(* Logix 5000 project; controller STAT 1756-L72 rev 20.12; software revision 20.04; part 3 of 34 *)

        [136]   // DELTA LVL NAOH TANK
        [137]   // PARAM CHUTE MAXI LVL NAOH
        [138]   // DELTA LVL H2SO4 TANK
        [139]   // PARAM CHUTE MAXI LVL H2SO4
        [140]   // MEMO LVL H2SO4
   N18 : DINT[120] := ([0] := 2829, [1] := 2829, [2] := 2845, [3] := 2845, [4] := 2829, [5] := 2845, [6] := 2845, [7] := 2845, [8] := 2829, [9] := 2829, [10] := 2845, [11] := 2845, [12] := 2845, [13] := 2845, [14] := 2845, [15] := 2845, [16] := 2845, [17] := 2845, [18] := 2829, [19] := 2820, [20] := 2845, [21] := 2845, [22] := 2845, [23] := 2845, [24] := 781, [25] := 2845, [26] := 781, [27] := 2845, [28] := 2829, [29] := 2820, [30] := 2845, [31] := 2829, [32] := 2829, [33] := 781, [34] := 2829, [35] := 781, [36] := 2829, [37] := 781, [38] := 2829, [39] := 2820, [40] := 2845, [41] := 781, [42] := 2829, [43] := 781, [44] := 2829, [45] := 2829, [46] := 2829, [47] := 2829, [48] := 2829, [49] := 2829, [50] := 2845, [51] := 2844, [52] := 2845, [53] := 2845, [54] := 2845, [55] := 2845, [56] := 2845, [57] := 2845, [58] := 2845, [59] := 2820,
        [60] := 2820, [61] := 2820, [62] := 2820, [63] := 2820, [64] := 2820, [65] := 2820, [66] := 2820, [67] := 2820, [68] := 2820, [69] := 2820, [70] := 2820, [71] := 2820, [72] := 2820, [73] := 2820, [74] := 2820, [75] := 2820, [76] := 2820, [77] := 2820, [78] := 2820, [79] := 2820, [80] := 2820, [105] := -1, [106] := -16369);
   N19 : DINT[80] := ([0] := 1779, [1] := 2603, [2] := 4997, [3] := 7884, [12] := 21845, [14] := 24576, [16] := 2048, [17] := 2048, [18] := 2048, [19] := 2048, [21] := -9, [50] := 128, [51] := 6, [52] := 300, [53] := -32768, [54] := 6, [55] := 300, [60] := 25600, [61] := 6, [62] := 300, [65] := 6, [66] := 300);
   N20 : DINT[80] := ([0] := 7500, [1] := 8000, [2] := 25600, [3] := 8000, [10] := -32768, [11] := 7500, [12] := 8000, [13] := 25600, [14] := 7500, [15] := 26214, [16] := 24576, [17] := 2048, [18] := 2048, [19] := 2048, [21] := -9, [50] := -32640, [51] := 6, [52] := 20, [54] := 7, [55] := 20, [60] := 17408, [62] := 20, [65] := 7, [66] := 20);
   N21 : DINT[80] := ([0] := 8000, [1] := 7000, [2] := 5000, [3] := 3000, [10] := -32768, [11] := 7500, [12] := 8000, [13] := 8000, [14] := 3000, [15] := 26214, [16] := 24576, [17] := 2048, [18] := 2048, [19] := 2048, [21] := -7, [50] := -32640, [51] := 6, [52] := 30, [54] := 7, [55] := 30, [60] := 1024, [62] := 30, [65] := 7, [66] := 30);
   N22 : DINT[80] := ([0] := 24000, [1] := 2000, [2] := 3000, [3] := 32000, [10] := -32768, [11] := 24000, [12] := 2000, [13] := 3000, [14] := 32000, [15] := 8738, [16] := 24576, [17] := 2048, [18] := 2048, [19] := 2048, [21] := -9, [50] := 128, [51] := 6, [52] := 40, [53] := -32768, [54] := 7, [55] := 40, [61] := 6, [62] := 40, [64] := 17408, [66] := 40);
   N23 : DINT[80] := ([0] := 5995, [1] := -2500, [2] := -2500, [3] := -2500, [10] := -32768, [11] := 32000, [12] := 21845, [14] := 24576, [16] := 2048, [17] := 2048, [18] := 2048, [19] := 2048, [21] := -9, [50] := -32640, [51] := 6, [52] := 150, [54] := 6, [55] := 150, [60] := 17408, [62] := 150, [65] := 6, [66] := 150);
        [0]   // DEBIET_PROMAG_33 debiet promag 33 0 -- 10 V
        [1]   // IST_FREQREG_PD1 istt freqreg pd1 0 -- 10 V
        [2]   // IST_FREQREG_PD2 istt freqreg pd2 0 -- 10 V
        [3]   // RESERVE_ANALO_IN reserve analoog ingang 0 tot 10V
   N24 : DINT[80] := ([2] := 234, [3] := 30000, [10] := -32768, [13] := 234, [14] := 30000, [15] := 8738, [16] := 24576, [17] := 2048, [18] := 2048, [19] := 2048, [21] := -9, [50] := -32640, [51] := 6, [52] := 160, [54] := 7, [55] := 160, [61] := 6, [62] := 160, [64] := 25600, [65] := 7, [66] := 160);
        [10]   // ??
        [11]   // SOLL_FREQREG_PD1 soll waarde pd1 0 - 10v
        [12]   // SOLL_FREQREG_PD2 soll freqreg pd2 0 -- 10v
   N26 : DINT[256] := ([0] := 3, [1] := 3, [2] := 7, [3] := 10, [4] := 300, [5] := 900, [6] := 20, [7] := 850, [8] := 60, [9] := 30, [20] := 2, [21] := 2, [22] := 7, [23] := 10, [24] := 300, [25] := 900, [26] := 20, [27] := 850, [28] := 60, [29] := 30, [36] := 1764, [42] := 15, [43] := 10, [44] := 30, [45] := 1200, [46] := 1800, [47] := 4500, [48] := 33, [49] := 5, [58] := 35, [62] := 15, [63] := 10, [64] := 30, [65] := 900, [66] := 1800, [67] := 4500, [68] := 33, [69] := 5, [82] := 20, [83] := 60, [84] := 60, [85] := 30, [86] := 120, [87] := 700, [88] := 20, [89] := 850, [90] := 60, [91] := 60, [102] := 15, [103] := 35, [104] := 10, [105] := 900, [106] := 1800, [107] := 4500, [108] := 35, [109] := 5, [122] := 15, [123] := 35, [124] := 10, [125] := 900,
        [126] := 1800, [127] := 4500, [128] := 35, [129] := 5, [132] := 10, [133] := 50, [134] := 10, [135] := 60, [136] := 7, [137] := 7, [138] := 960, [142] := 10, [143] := 50, [144] := 10, [145] := 60, [146] := 7, [148] := 900, [152] := 10, [153] := 50, [154] := 10, [155] := 60, [156] := 7, [158] := 960, [172] := 10, [173] := 1, [174] := 1, [175] := 9000, [176] := 600, [177] := 1, [178] := 1, [179] := 1800, [182] := 20, [183] := 1, [184] := 1, [185] := 18000, [186] := 600, [187] := 1, [188] := 1, [189] := 1800, [190] := 1, [191] := 1, [192] := 5, [193] := 1, [194] := 1, [195] := 1800, [196] := 600, [197] := 1, [198] := 1, [199] := 1800, [200] := 1, [201] := 2000, [202] := 600, [203] := 1, [204] := 1, [205] := 1800, [206] := 600);
        [0]   // SOLL_ST_SPOELTFB75_1 Soll stap spoel TFB 75-1 ingave via visualisatie
        [1]   // IST_ST_SPOELTFB75_1 Ist stap spoel TFB 75-1 ingave via visualisatie
        [2]   // SOLL_TIJD_ST_1 Soll tijd stap 1 spoel TFB75 -1 Afsluiten filter
        [3]   // SOLL_TIJD_ST_2 Soll tijd stap 2 spoel TFB75 -1 Aflaten water
        [4]   // SOLL_TIJD_ST_3 Soll tijd stap 3 spoel TFB75 -1 luchtspoeling
        [5]   // SOLL_TIJD_ST_4 Soll tijd stap 4 spoel TFB75 -1 rustpauze
        [6]   // SOLL_TIJD_ST_5 Soll tijd stap 5 spoel TFB75 -1 Waterspoeling
        [7]   // SOLL_TIJD_ST_6 Soll tijd stap 6 spoel TFB75 -1 Rustpauze
        [8]   // SOLL_TIJD_ST_7 Soll tijd stap 7 spoel TFB75 -1 Openen filter
        [10]   // SOLL_TIJD_ST_8
        [11]   // SOLL_TIJD_ST_9
        [12]   // SOLL_TIJD_ST_10
        [13]   // SOLL_TIJD_ST_11
        [14]   // SOLL_TIJD_ST_12
        [15]   // SOLL_TIJD_ST_13
        [16]   // SOLL_TIJD_ST_14
        [17]   // SOLL_TIJD_ST_15
        [18]   // SOLL_TIJD_ST_16
        [20]   // SOLL_ST_SPOETFB75_2
        [21]   // IST_ST_SPOETFB75_2
        [22]   // SOLL_TIJD_STA_1_1
        [23]   // SOLL_TIJD_STA_2_2
        [24]   // SOLL_TIJD_STA_3_2
        [25]   // SOLL_TIJD_STA_4_2
        [26]   // SOLL_TIJD_STA_5_2
        [27]   // SOLL_TIJD_STA_6_2
        [28]   // SOLL_TIJD_STA_7_2
   N28 : DINT[80] := ([0] := 10249, [1] := 10249, [2] := 10249, [3] := 10249, [10] := -32768, [11] := 32000, [12] := 26214, [14] := 24576, [16] := 2048, [17] := 2048, [18] := 2048, [19] := 2048, [21] := -11, [22] := -11, [50] := 128, [51] := 6, [52] := 150, [53] := -32768, [54] := 6, [55] := 150, [60] := 4096, [62] := 150, [63] := -11, [66] := 150, [67] := -11);
   N7 : DINT[255] := ([0] := 7825, [1] := 3859, [2] := 8045, [3] := -2501, [12] := 21845, [14] := 24576, [16] := 2048, [17] := 2048, [18] := 2048, [19] := 2048, [21] := -9, [33] := 16383, [40] := 45, [41] := 40, [42] := 35, [43] := 50, [44] := 45, [45] := 35, [50] := -32640, [51] := 6, [52] := 260, [54] := 6, [55] := 260, [60] := 17408, [62] := 260, [65] := 6, [66] := 260, [70] := 80, [71] := 38, [72] := 78, [92] := 6, [100] := 15900, [101] := 15900, [110] := -32768, [111] := 4, [186] := 16, [190] := 7, [191] := 1, [197] := 2, [198] := 8, [199] := 96, [200] := 22, [201] := 1564, [211] := 1028, [225] := 1048576, [234] := 31233);
        [70]   // aux LEVEL TANK RECUP L3
        [71]   // n7:71
        [90]   // ?
        [97]   // ?
        [98]   // ?
        [111]   // HULPWOORD_N1
        [112]   // HULPWOORD_N2
        [113]   // HULPWOORD_N3
        [114]   // HULPWOORD_N4
        [115]   // HULPWOORD_N5
        [190]   // PRIORITE DEFAUT
        [191]   // defaut niv 2
        [197]   // NOMBRE DEFAUT EXISTANT ACQUITE
        [198]   // NOMBRE NOUVEAU DEFAUT
        [199].0   // arret entretien
        [199].1   // acquit defaut
        [199].5   // new defaut
        [199].6   // ancien defaut present
        [200].0   // PMP ETANG EN DEF
        [200].1   // no flow pumping from etang
        [200].2   // FLOW TOO LOW Q1
        [200].3   // LEVEL PRETREATED TOO HIGH
        [200].4   // LEVEL LOW PRETREATED WATER WARNING
        [200].5   // LEVEL LOW PRETREATED WATER
        [200].6   // ANORMAL EMPTYING PRETREATED WATER TANK
        [200].7   // 2 pump pretreated tank out of order P3&P4
        [200].8   // no flow pumping from PRETREATED WATER TANK
        [200].9   // FLOW TOO LOW Q2
        [200].11   // recup water tank L1 too high
        [200].12   // PMP RECUP L1 OUT OF ORDER
        [200].13   // recup water tank L2 too high
        [200].14   // PMP RECUP L2 OUT OF ORDER
        [200].15   // recup water tank L3 too high
        [201].0   // PMP RECUP L3 OUT OF ORDER
        [201].1   // recup water tank L4 too high
        [201].2   // PMP RECUP L4 OUT OF ORDER
        [201].3   // LEVEL NAOH TOO HIGH
        [201].4   // ANORMAL LEVEL DECREASE naoh TANK
        [201].5   // LACK DETECTIE NAOH
        [201].6   // LEVEL H2SO4 TOO HIGH
        [201].7   // ANORMAL LEVEL DECREASE H2SO4 TANK
        [201].8   // LACK DETECTIE H2SO4
        [201].9   // defaut niveau vijver trop bas
        [201].10   // defaut niveau puisard ligne 4
        [201].11   // defaut vanne position eau ville
        [210].0   // PMP ETANG EN DEF
        [210].1   // no flow pumping from etang
        [210].2   // FLOW TOO LOW Q1
        [210].3   // LEVEL PRETREATED TOO HIGH
        [210].4   // LEVEL LOW PRETREATED WATER WARNING
        [210].5   // LEVEL LOW PRETREATED WATER
        [210].6   // ANORMAL EMPTYING PRETREATED WATER TANK
        [210].7   // 2 pump pretreated tank out of order P3&P4
        [210].8   // no flow pumping from PRETREATED WATER TANK
        [210].9   // FLOW TOO LOW Q2
        [210].11   // recup water tank L1 too high
        [210].12   // PMP RECUP L1 OUT OF ORDER
        [210].13   // recup water tank L2 too high
        [210].14   // PMP RECUP L2 OUT OF ORDER
        [210].15   // recup water tank L3 too high
        [211].0   // PMP RECUP L3 OUT OF ORDER
        [211].1   // recup water tank L4 too high
        [211].2   // PMP RECUP L4 OUT OF ORDER
        [211].3   // LEVEL NAOH TOO HIGH
        [211].4   // ANORMAL LEVEL DECREASE naoh TANK
        [211].5   // LACK DETECTIE NAOH
        [211].6   // LEVEL H2SO4 TOO HIGH
        [211].7   // ANORMAL LEVEL DECREASE H2SO4 TANK
        [211].8   // LACK DETECTIE H2SO4
        [211].9   // defaut niveau vijver trop bas
        [211].11   // memo defaut vanne position eau ville
   N7_70 : REAL := 80.299995;
   N7_71 : REAL := 99.04;
   N7_72 : REAL := 1561.2001;
   naohL1VA4 : BOOL;
   naohL2VA4 : BOOL;
   O1 : INT[32] := ([6] := 2#1000_0000_0000_0000, [11] := 2#0000_0000_0000_0011, [12] := 2#0000_0000_0000_0010, [20] := 2#0000_0110_0000_0110);
   O11 : INT[2] := ([0] := 2#0101_1000_0001_1010, [1] := 2#1011_0000_0000_0110);
   O11_000_Bit00 : ALIAS FOR O11[0].0;   // Motor P11 lijn 1 P11_LIJN_1
   O11_000_Bit01 : ALIAS FOR O11[0].1;   // Motor P12 lijn 1 P12_LIJN_1
   O11_000_Bit02 : ALIAS FOR O11[0].2;   // Motor P13 lijn 2 P13_LIJN_2
   O11_000_Bit03 : ALIAS FOR O11[0].3;   // Motor P14 lijn 2 P14_LIJN_2
   O11_000_Bit04 : ALIAS FOR O11[0].4;   // Motor P15 lijn 3 P15_LIJN_3
   O11_000_Bit05 : ALIAS FOR O11[0].5;   // Motor P16 lijn 3 P16_LIJN_3
   O11_000_Bit06 : ALIAS FOR O11[0].6;   // Motor P17 lijn 4 P17_LIJN_4
   O11_000_Bit07 : ALIAS FOR O11[0].7;   // Motor P18 lijn 4 P18_LIJN_4
   O11_000_Bit08 : ALIAS FOR O11[0].8;   // Pomp voeding osmose 1 lijn PRO1_OSMO1_LIJN
   O11_000_Bit09 : ALIAS FOR O11[0].9;   // Pomp voeding osmose 1 driehoek PRO1_OSMO1_DRIE
   O11_000_Bit10 : ALIAS FOR O11[0].10;   // Pomp voeding osmose 1 ster PRO1_OSMO1_STER
   O11_000_Bit11 : ALIAS FOR O11[0].11;   // Pomp voeding osmose 2 lijn PRO1_OSMO2_LIJN
   O11_000_Bit12 : ALIAS FOR O11[0].12;   // Pomp voeding osmose 2 driehoek PRO1_OSMO2_DRIE
   O11_000_Bit13 : ALIAS FOR O11[0].13;   // Pomp voeding osmose 2 ster PRO1_OSMO2_STER
   O11_000_Bit14 : ALIAS FOR O11[0].14;   // pomp 21 kuip az P21_KUIP_AZ_LIJN
   O11_000_Bit15 : ALIAS FOR O11[0].15;   // pomp p21 kuip az driehoek P21_KUIP_AZ_DRIE
   O11_001_Bit00 : ALIAS FOR O11[1].0;   // pomp p21 kuip az ster P21_KUIP_AZ_STER
   O11_001_Bit01 : ALIAS FOR O11[1].1;   // pomp p22 kuip az lijn P22_KUIP_AZ_LIJN
   O11_001_Bit02 : ALIAS FOR O11[1].2;   // pomp p22 kuip az drie P22_KUIP_AZ_DRIE
   O11_001_Bit03 : ALIAS FOR O11[1].3;   // pomp p22 kuip az ster P22_KUIP_AZ_STER
   O11_001_Bit04 : ALIAS FOR O11[1].4;   // Voedingspomp osmose 3 in lijn PRO3_OSMOSE3_LIJN
   O11_001_Bit05 : ALIAS FOR O11[1].5;   // Voedingspomp osmose 3 in drie PRO3_OSMOSE3_DRIE
   O11_001_Bit06 : ALIAS FOR O11[1].6;   // Voedingspomp osmose 3 in ster PRO3_OSMOSE3_STER
   O11_001_Bit07 : ALIAS FOR O11[1].7;   // reinigingspomp membraam P21_REINIG
   O11_001_Bit08 : ALIAS FOR O11[1].8;   // ventilator s1 S1_VENT
   O11_001_Bit09 : ALIAS FOR O11[1].9;   // pomp voeding drive 1 in lijn P3_FAB_LIJN
   O11_001_Bit10 : ALIAS FOR O11[1].10;   // pomp debloquage 1 P3 P3_FAB_DRIE
   O11_001_Bit11 : ALIAS FOR O11[1].11;   // pomp voeding fab1 in ster P3_FAB_STER
   O11_001_Bit12 : ALIAS FOR O11[1].12;   // pomp voeding fabriek 2 in lijn P4_FAB_LIJN
   O11_001_Bit13 : ALIAS FOR O11[1].13;   // deverouillage drive P4 P4_FAB_DRIE
   O11_001_Bit14 : ALIAS FOR O11[1].14;   // reserve P4_FAB_STER
   O11_001_Bit15 : ALIAS FOR O11[1].15;   // spoelpomp filters dubbele media P5_SPOEL
   O12 : INT[2] := ([0] := 2#1100_1000_1001_1000, [1] := 2#0111_0100_1101_0000);
   O12_000_Bit00 : ALIAS FOR O12[0].0;   // spoelpomp filters dubbele media P6_SPOEL
   O12_000_Bit01 : ALIAS FOR O12[0].1;   // pomp pompen uit kelder P23_KELDER
   O12_000_Bit02 : ALIAS FOR O12[0].2;   // pomp pompen uit kelder P24_KELDER
   O12_000_Bit03 : ALIAS FOR O12[0].3;   // motor ag1 mixer krimp neutralisatie AG1_MIXER_KRIMP
   O12_000_Bit04 : ALIAS FOR O12[0].4;   // Motor doseerpomp acide pd3 PD3_DOS_ACIDE
   O12_000_Bit05 : ALIAS FOR O12[0].5;   // Motor doseerpomp acide pd4 PD4_DOS_ACIDE
   O12_000_Bit06 : ALIAS FOR O12[0].6;   // Motor doseerpomp acide pd5 soude PD5_DOS_SOUDE
   O12_000_Bit07 : ALIAS FOR O12[0].7;   // Motor doseerpomp acide pd6 soude PD6_DOS_SOUDE
   O12_000_Bit08 : ALIAS FOR O12[0].8;   // pomp ag2 mixer vat 1 AG2_MIXER_VAT1
   O12_000_Bit09 : ALIAS FOR O12[0].9;   // pomp ag3 mixer vat 2 AG3_MIXER_VAT2
   O12_000_Bit10 : ALIAS FOR O12[0].10;   // pomp pd7 doseerpomp floculaat PD7_DOSEER_FLOCU
   O12_000_Bit11 : ALIAS FOR O12[0].11;   // pomp pd8 doseerpomp floculaat PD8_DOSEER_FLOCU
   O12_000_Bit12 : ALIAS FOR O12[0].12;   // Motor P19a zuiveringspomp controleweger P19_ZUIVERP
   O12_000_Bit13 : ALIAS FOR O12[0].13;   // Motor P20 zuiveringspomp controleweger P20_ZUIVERP
   O12_000_Bit14 : ALIAS FOR O12[0].14;   // Motor Pm1 recerculatiepomp ingang 1 decanter PM1_RECER_DEC1
   O12_000_Bit15 : ALIAS FOR O12[0].15;   // Motor Pm2 recerculatiepomp ingang 2 decanter PM2_RECER_DEC2
   O12_001_Bit00 : ALIAS FOR O12[1].0;   // Motor Pm3 evacuatiepomp ingang 1 decanter PM3_EVACU_IN_1
   O12_001_Bit01 : ALIAS FOR O12[1].1;   // Motor Pm4 evacuatiepomp ingang 2 decanter PM4_EVACU_IN_2
   O12_001_Bit02 : ALIAS FOR O12[1].2;   // Motor P25 pekel P25_POMP_PEKEL
   O12_001_Bit03 : ALIAS FOR O12[1].3;   // Motor P7 voedingspomp omgekeerde osmose 1 P7_OSMOSE_1
   O12_001_Bit04 : ALIAS FOR O12[1].4;   // Motor P8 voedingspomp omgekeerde osmose 2 P8_OSMOSE_2
   O12_001_Bit05 : ALIAS FOR O12[1].5;   // Motor P9 voedingspomp omgekeerde osmose 3 P9_OSMOSE_3
   O12_001_Bit06 : ALIAS FOR O12[1].6;   // TFB1_1_EV1 TFB1_1_EV1
   O12_001_Bit07 : ALIAS FOR O12[1].7;   // TFB1_1_EV2 TFB1_1_EV2
   O12_001_Bit08 : ALIAS FOR O12[1].8;   // TFB1_2_EV3 TFB1_2_EV3
   O12_001_Bit09 : ALIAS FOR O12[1].9;   // TFB1_2_EV4 TFB1_2_EV4
   O12_001_Bit10 : ALIAS FOR O12[1].10;   // TFB1_2_EV10 TFB1_2_EV10
   O12_001_Bit11 : ALIAS FOR O12[1].11;   // TFB1_EV9 TFB1_EV9
   O12_001_Bit12 : ALIAS FOR O12[1].12;   // TFB1_2_EV5 TFB1_2_EV5
   O12_001_Bit13 : ALIAS FOR O12[1].13;   // TFB1_2_EV6 TFB1_2_EV6
   O12_001_Bit14 : ALIAS FOR O12[1].14;   // STFA1_EV1 STFA1_EV1
   O12_001_Bit15 : ALIAS FOR O12[1].15;   // STFA1_EV2 STFA1_EV2
   O13 : INT[2] := ([0] := 2#0000_0000_0000_1000, [1] := 2#0001_0000_0000_0000);
   O13_000_Bit00 : ALIAS FOR O13[0].0;   // STFA1_EV3 STFA1_EV3
   O13_000_Bit01 : ALIAS FOR O13[0].1;   // STFA1_EV4 STFA1_EV4
   O13_000_Bit02 : ALIAS FOR O13[0].2;   // STFA1_EV5 STFA1_EV5
   O13_000_Bit03 : ALIAS FOR O13[0].3;   // STFA1_EV6 STFA1_EV6
   O13_000_Bit06 : ALIAS FOR O13[0].6;   // PULS_DOSEER_PD3
   O13_000_Bit07 : ALIAS FOR O13[0].7;   // PULS_DOSEER_PD4
   O13_000_Bit08 : ALIAS FOR O13[0].8;   // PULS_DOSEER_PD5
   O13_000_Bit09 : ALIAS FOR O13[0].9;   // PULS_DOSEER_PD6
   O13_000_Bit12 : ALIAS FOR O13[0].12;   // STFA2_EV1 STFA2_EV1
   O13_000_Bit13 : ALIAS FOR O13[0].13;   // STFA2_EV2 STFA2_EV2
   O13_000_Bit14 : ALIAS FOR O13[0].14;   // STFA2_EV3 STFA2_EV3
   O13_000_Bit15 : ALIAS FOR O13[0].15;   // STFA2_EV4 STFA2_EV4
   O13_001_Bit0 : ALIAS FOR O13[1].0;   // STFA2_EV5 STFA2_EV5
   O13_001_Bit1 : ALIAS FOR O13[1].1;   // STFA2_EV6 STFA2_EV6
   O13_001_Bit10 : ALIAS FOR O13[1].10;   // TFB1_2_EV7 TFB1_2_EV7
   O13_001_Bit11 : ALIAS FOR O13[1].11;   // TFB1_2_EV8 TFB1_2_EV8
   O13_001_Bit12 : ALIAS FOR O13[1].12;   // TFB1_2_EV11 TFB1_2_EV11
   O13_001_Bit13 : ALIAS FOR O13[1].13;   // vanne eau de ville
   O14 : INT[2] := ([0] := 2#1000_0000_0000_0000, [1] := 2#0011_0000_0010_0010);
   O14_000_Bit14 : ALIAS FOR O14[0].14;   // STFA3_EV1 STFA3_EV1
   O14_000_Bit15 : ALIAS FOR O14[0].15;   // STFA3_EV2 STFA3_EV2
   O14_001_Bit00 : ALIAS FOR O14[1].0;   // STFA3_EV3 STFA3_EV3
   O14_001_Bit01 : ALIAS FOR O14[1].1;   // STFA3_EV4 STFA3_EV4
   O14_001_Bit02 : ALIAS FOR O14[1].2;   // STFA3_EV5 STFA3_EV5
   O14_001_Bit03 : ALIAS FOR O14[1].3;   // STFA3_EV6 STFA3_EV6
   O14_001_Bit04 : ALIAS FOR O14[1].4;   // kalxon out NAOH
   O14_001_Bit05 : ALIAS FOR O14[1].5;   // lampe out NAOH
   O14_001_Bit06 : ALIAS FOR O14[1].6;   // klaxon out H2SO4
   O14_001_Bit07 : ALIAS FOR O14[1].7;   // lampe H2SO4
   O14_001_Bit08 : ALIAS FOR O14[1].8;   // klaxon out ZOUT
   O14_001_Bit09 : ALIAS FOR O14[1].9;   // lampe ZOUT
   O14_001_Bit12 : ALIAS FOR O14[1].12;   // RO1_EV1 RO1_EV1
   O14_001_Bit13 : ALIAS FOR O14[1].13;   // RO1_EV2 RO1_EV2
   O15 : INT[2] := ([1] := 2#0000_0000_1000_0000);
   O15_000_Bit00 : ALIAS FOR O15[0].0;   // RO2_EV1 RO2_EV1
   O15_000_Bit01 : ALIAS FOR O15[0].1;   // RO2_EV2 RO2_EV2
   O15_000_Bit04 : ALIAS FOR O15[0].4;   // RO3_EV1 RO3_EV1
   O15_000_Bit05 : ALIAS FOR O15[0].5;   // RO3_EV2 RO3_EV2
   O15_000_Bit09 : ALIAS FOR O15[0].9;   // CLEAN_V11 CLEAN_V11
   O15_000_Bit10 : ALIAS FOR O15[0].10;   // CLEAN_V12 CLEAN_V12
   O15_000_Bit11 : ALIAS FOR O15[0].11;   // CLEAN_V13 CLEAN_V13
   O15_000_Bit12 : ALIAS FOR O15[0].12;   // CLEAN_V14 CLEAN_V14
   O15_000_Bit13 : ALIAS FOR O15[0].13;   // CLEAN_V21 CLEAN_V21
   O15_000_Bit14 : ALIAS FOR O15[0].14;   // CLEAN_V22 CLEAN_V22
   O15_000_Bit15 : ALIAS FOR O15[0].15;   // CLEAN_V23 CLEAN_V23
   O15_001_Bit00 : ALIAS FOR O15[1].0;   // CLEAN_V24 CLEAN_V24
   O15_001_Bit01 : ALIAS FOR O15[1].1;   // CLEAN_V3 CLEAN_V3
   O15_001_Bit06 : ALIAS FOR O15[1].6;   // EV2 EV2
   O15_001_Bit07 : ALIAS FOR O15[1].7;   // EV3 EV3
   O15_001_Bit08 : ALIAS FOR O15[1].8;   // EV4 EV4
   O15_001_Bit09 : ALIAS FOR O15[1].9;   // EV5 EV5
   O15_001_Bit10 : ALIAS FOR O15[1].10;   // EV6 EV6
   O15_001_Bit11 : ALIAS FOR O15[1].11;   // EV7 EV7
   O15_001_Bit13 : ALIAS FOR O15[1].13;   // TFB2_1_EV1 TFB2_1_EV1
   O15_001_Bit14 : ALIAS FOR O15[1].14;   // TFB2_1_EV2 TFB2_1_EV2
   O15_001_Bit15 : ALIAS FOR O15[1].15;   // TFB2_1_EV3 TFB2_1_EV3
   O16 : INT[2] := ([0] := 2#1001_0100_0000_1001, [1] := 2#1100_0000_0000_0000);
        [0].4   // vanne soude de stock
        [0].3   // vanne ibt acide de stock
   O16_000_Bit00 : ALIAS FOR O16[0].0;   // COMMANDE VANNE ALIBERT
   O16_000_Bit01 : ALIAS FOR O16[0].1;   // vanne pmp puit 3
   O16_000_Bit02 : ALIAS FOR O16[0].2;   // vanne pmp puit 2
   O16_000_Bit03 : ALIAS FOR O16[0].3;
   O16_000_Bit09 : ALIAS FOR O16[0].9;   // LAMP_P17_AAN
   O16_000_Bit10 : ALIAS FOR O16[0].10;   // LAMP_P17_UIT
   O16_000_Bit11 : ALIAS FOR O16[0].11;   // LAMP_P18_AAN
   O16_000_Bit12 : ALIAS FOR O16[0].12;   // LAMP_P18_UIT
   O16_000_Bit15 : ALIAS FOR O16[0].15;   // LAMP_PRO1_AAN
   O16_001_Bit00 : ALIAS FOR O16[1].0;   // LAMP_PRO1_UIT
   O16_001_Bit01 : ALIAS FOR O16[1].1;   // LAMP_PRO2_AAN
   O16_001_Bit02 : ALIAS FOR O16[1].2;   // LAMP_PRO2_UIT
   O16_001_Bit03 : ALIAS FOR O16[1].3;   // LAMP_P21_AAN
   O16_001_Bit04 : ALIAS FOR O16[1].4;   // LAMP_P21_UIT
   O16_001_Bit05 : ALIAS FOR O16[1].5;   // LAMP_P22_AAN
   O16_001_Bit06 : ALIAS FOR O16[1].6;   // LAMP_P22_UIT
   O16_001_Bit07 : ALIAS FOR O16[1].7;   // LAMP_PRO3_AAN
   O16_001_Bit08 : ALIAS FOR O16[1].8;   // LAMP_PRO3_UIT
   O16_001_Bit09 : ALIAS FOR O16[1].9;   // LAMP_P21_REINIG_AAN
   O16_001_Bit10 : ALIAS FOR O16[1].10;   // LAMP_P21_REINIG_UIT
   O16_001_Bit11 : ALIAS FOR O16[1].11;   // LAMP_VENT_S1_AAN
   O16_001_Bit12 : ALIAS FOR O16[1].12;   // LAMP_VENT_S1_UIT
   O16_001_Bit13 : ALIAS FOR O16[1].13;   // LAMP_P3_AAN
   O16_001_Bit14 : ALIAS FOR O16[1].14;   // LAMP_P3_UIT
   O16_001_Bit15 : ALIAS FOR O16[1].15;   // LAMP_P4_AAN
   O17 : INT[2] := ([0] := 2#0000_0010_0000_0000, [1] := 2#0010_1010_0001_0010);
   O17_000_Bit00 : ALIAS FOR O17[0].0;   // LAMP_P4_UIT
   O17_000_Bit01 : ALIAS FOR O17[0].1;   // LAMP_P5_AAN
   O17_000_Bit02 : ALIAS FOR O17[0].2;   // LAMP_P5_UIT
   O17_000_Bit03 : ALIAS FOR O17[0].3;   // LAMP_P6_AAN
   O17_000_Bit04 : ALIAS FOR O17[0].4;   // LAMP_P6_UIT
   O17_000_Bit05 : ALIAS FOR O17[0].5;   // LAMP_P23_AAN
   O17_000_Bit06 : ALIAS FOR O17[0].6;   // LAMP_P23_UIT
   O17_000_Bit07 : ALIAS FOR O17[0].7;   // LAMP_P24_AAN
   O17_000_Bit08 : ALIAS FOR O17[0].8;   // LAMP_P24_UIT
   O17_000_Bit09 : ALIAS FOR O17[0].9;   // LAMP_AG1_AAN
   O17_000_Bit10 : ALIAS FOR O17[0].10;   // LAMP_AG1_UIT
   O17_000_Bit11 : ALIAS FOR O17[0].11;   // LAMP_AG2_AAN
   O17_000_Bit12 : ALIAS FOR O17[0].12;   // LAMP_AG2_UIT
   O17_000_Bit13 : ALIAS FOR O17[0].13;   // LAMP_AG3_AAN
   O17_000_Bit14 : ALIAS FOR O17[0].14;   // LAMP_AG3_UIT
   O17_000_Bit15 : ALIAS FOR O17[0].15;   // LAMP_PD7_AAN
   O17_001_Bit00 : ALIAS FOR O17[1].0;   // LAMP_PD7_UIT
   O17_001_Bit01 : ALIAS FOR O17[1].1;   // LAMP_PD8_AAN
   O17_001_Bit02 : ALIAS FOR O17[1].2;   // LAMP_PD8_UIT
   O17_001_Bit03 : ALIAS FOR O17[1].3;   // LAMP_P19A_AAN
   O17_001_Bit04 : ALIAS FOR O17[1].4;   // LAMP_P19A_UIT
   O17_001_Bit05 : ALIAS FOR O17[1].5;   // LAMP_P19B_AAN
   O17_001_Bit06 : ALIAS FOR O17[1].6;   // LAMP_P19B_UIT
   O17_001_Bit09 : ALIAS FOR O17[1].9;   // LAMP_P25_AAN
   O17_001_Bit10 : ALIAS FOR O17[1].10;   // LAMP_P25_UIT
   O17_001_Bit11 : ALIAS FOR O17[1].11;   // LAMP_PM1_AAN
   O17_001_Bit12 : ALIAS FOR O17[1].12;   // LAMP_PM1_UIT
   O17_001_Bit13 : ALIAS FOR O17[1].13;   // LAMP_PM2_AAN
   O17_001_Bit14 : ALIAS FOR O17[1].14;   // LAMP_PM2_UIT
   O17_001_Bit15 : ALIAS FOR O17[1].15;   // LAMP_PM3_AAN
   O18 : INT[2] := ([0] := 2#0000_0010_0000_0000, [1] := 2#0000_0000_0001_0100);
   O18_000_Bit00 : ALIAS FOR O18[0].0;   // LAMP_PM3_UIT
   O18_000_Bit01 : ALIAS FOR O18[0].1;   // LAMP_PM4_AAN
   O18_000_Bit02 : ALIAS FOR O18[0].2;   // LAMP_PM4_UIT
   O18_000_Bit07 : ALIAS FOR O18[0].7;   // LAMP_P7_AAN
   O18_000_Bit08 : ALIAS FOR O18[0].8;   // LAMP_P7_UIT
   O18_000_Bit09 : ALIAS FOR O18[0].9;   // LAMP_P8_AAN
   O18_000_Bit10 : ALIAS FOR O18[0].10;   // LAMP_P8_UIT
   O18_000_Bit11 : ALIAS FOR O18[0].11;   // LAMP_P9_AAN
   O18_000_Bit12 : ALIAS FOR O18[0].12;   // LAMP_P9_UIT
   O18_001_Bit00 : ALIAS FOR O18[1].0;   // pompe 1 puisard ligne 4
   O18_001_Bit01 : ALIAS FOR O18[1].1;   // pompe 2 puisard ligne 4
   O18_001_Bit02 : ALIAS FOR O18[1].2;   // pmp put 2
   O18_001_Bit03 : ALIAS FOR O18[1].3;   // PMP PUT over
   O18_001_Bit04 : ALIAS FOR O18[1].4;   // PMP PUT 1
   O18_001_Bit05 : ALIAS FOR O18[1].5;   // pmp vijver IWM
   O18_001_Bit06 : ALIAS FOR O18[1].6;
   O18_001_Bit07 : ALIAS FOR O18[1].7;   // pomp pompen uit kelder p23
   O18_001_Bit08 : ALIAS FOR O18[1].8;   // pomp pompen uit kelder p24
   O1_006_Bit15 : ALIAS FOR O1[6].15;
   O1_011_Bit00 : ALIAS FOR O1[11].0;
   O1_011_Bit01 : ALIAS FOR O1[11].1;
   O1_011_Bit02 : ALIAS FOR O1[11].2;
   O1_011_Bit03 : ALIAS FOR O1[11].3;
   O1_011_Bit04 : ALIAS FOR O1[11].4;
   O1_011_Bit05 : ALIAS FOR O1[11].5;
   O1_011_Bit06 : ALIAS FOR O1[11].6;
   O1_011_Bit07 : ALIAS FOR O1[11].7;
   O1_011_Bit08 : ALIAS FOR O1[11].8;
   O1_011_Bit09 : ALIAS FOR O1[11].9;
   O1_011_Bit10 : ALIAS FOR O1[11].10;
   O1_012_Bit01 : ALIAS FOR O1[12].1;
   O1_012_Bit02 : ALIAS FOR O1[12].2;
   O1_012_Bit03 : ALIAS FOR O1[12].3;
   O1_012_Bit04 : ALIAS FOR O1[12].4;
   O1_012_Bit05 : ALIAS FOR O1[12].5;
   O1_012_Bit06 : ALIAS FOR O1[12].6;
   O1_012_Bit07 : ALIAS FOR O1[12].7;
   O1_012_Bit08 : ALIAS FOR O1[12].8;
   O1_012_Bit09 : ALIAS FOR O1[12].9;
   O1_012_Bit10 : ALIAS FOR O1[12].10;
   O1_020_Bit00 : ALIAS FOR O1[20].0;
   O1_020_Bit01 : ALIAS FOR O1[20].1;
   O1_020_Bit02 : ALIAS FOR O1[20].2;
   O1_020_Bit03 : ALIAS FOR O1[20].3;
   O1_020_Bit08 : ALIAS FOR O1[20].8;
   O1_020_Bit09 : ALIAS FOR O1[20].9;
   O1_020_Bit10 : ALIAS FOR O1[20].10;
   O1_020_Bit11 : ALIAS FOR O1[20].11;
   O1_021_Bit00 : ALIAS FOR O1[21].0;
   O1_021_Bit01 : ALIAS FOR O1[21].1;
   O1_021_Bit02 : ALIAS FOR O1[21].2;
   O1_021_Bit03 : ALIAS FOR O1[21].3;
   O1_021_Bit08 : ALIAS FOR O1[21].8;
   O1_021_Bit09 : ALIAS FOR O1[21].9;
   O20 : INT[8] := ([0] := 2#0000_1011_0000_1101, [1] := 2#0000_1011_0000_1101, [2] := 2#0000_1011_0001_1101, [3] := 2#0000_1011_0001_1101, [4] := 2#0000_1011_0000_1101, [5] := 2#0000_1011_0001_1101, [6] := 2#0000_1011_0001_1101, [7] := 2#0000_1011_0001_1101);
   O20_000 : ALIAS FOR O20[0];
   O20_001 : ALIAS FOR O20[1];
   O20_002 : ALIAS FOR O20[2];
   O20_003 : ALIAS FOR O20[3];
   O20_004 : ALIAS FOR O20[4];
   O20_005 : ALIAS FOR O20[5];
   O20_006 : ALIAS FOR O20[6];
   O20_007 : ALIAS FOR O20[7];
   O21 : INT[8] := ([0] := 2#0000_1011_0001_1101, [1] := 2#0000_1011_0001_1101, [2] := 2#0000_1011_0001_1101, [3] := 2#0000_1011_0001_1101, [4] := 2#0000_1011_0001_1101, [5] := 2#0000_1011_0001_1101, [6] := 2#0000_1011_0001_1101, [7] := 2#0000_1011_0001_1101);
   O21_000 : ALIAS FOR O21[0];
   O21_001 : ALIAS FOR O21[1];
   O21_002 : ALIAS FOR O21[2];
   O21_003 : ALIAS FOR O21[3];
   O21_004 : ALIAS FOR O21[4];
   O21_005 : ALIAS FOR O21[5];
   O21_006 : ALIAS FOR O21[6];
   O21_007 : ALIAS FOR O21[7];
   O22 : INT[8] := ([0] := 2#0000_1011_0001_1101, [1] := 2#0000_1011_0001_1101, [2] := 2#0000_1011_0001_1101, [3] := 2#0000_1011_0001_1101, [4] := 2#0000_0011_0000_1101, [5] := 2#0000_1011_0001_1101, [6] := 2#0000_0011_0000_1101, [7] := 2#0000_1011_0001_1101);
   O22_000 : ALIAS FOR O22[0];
   O22_000_Bit04 : ALIAS FOR O22[0].4;
   O22_001 : ALIAS FOR O22[1];
   O22_002 : ALIAS FOR O22[2];
   O22_003 : ALIAS FOR O22[3];
   O22_004 : ALIAS FOR O22[4];
   O22_005 : ALIAS FOR O22[5];
   O22_006 : ALIAS FOR O22[6];
   O22_007 : ALIAS FOR O22[7];
   O23 : INT[8] := ([0] := 2#0000_1011_0001_1101, [1] := 2#0000_1011_0000_1101, [2] := 2#0000_1011_0000_1101, [3] := 2#0000_0011_0000_1101, [4] := 2#0000_1011_0000_1101, [5] := 2#0000_1011_0000_1101, [6] := 2#0000_1011_0000_1101, [7] := 2#0000_0011_0000_1101);
   O23_000 : ALIAS FOR O23[0];
   O23_001 : ALIAS FOR O23[1];
   O23_002 : ALIAS FOR O23[2];
   O23_003 : ALIAS FOR O23[3];
   O23_004 : ALIAS FOR O23[4];
   O23_005 : ALIAS FOR O23[5];
   O23_006 : ALIAS FOR O23[6];
   O23_007 : ALIAS FOR O23[7];
   O24 : INT[8] := ([0] := 2#0000_1011_0001_1101, [1] := 2#0000_0011_0000_1101, [2] := 2#0000_1011_0000_1101, [3] := 2#0000_0011_0000_1101, [4] := 2#0000_1011_0000_1101, [5] := 2#0000_1011_0000_1101, [6] := 2#0000_1011_0000_1101, [7] := 2#0000_1011_0000_1101);
   O24_000 : ALIAS FOR O24[0];
   O24_001 : ALIAS FOR O24[1];
   O24_002 : ALIAS FOR O24[2];
   O24_003 : ALIAS FOR O24[3];
   O24_004 : ALIAS FOR O24[4];
   O24_005 : ALIAS FOR O24[5];
   O24_006 : ALIAS FOR O24[6];
   O24_007 : ALIAS FOR O24[7];
   O25 : INT[8] := ([0] := 2#0000_1011_0001_1101, [1] := 2#0000_1011_0001_1100, [2] := 2#0000_1011_0001_1101, [3] := 2#0000_1011_0001_1101, [4] := 2#0000_1011_0001_1101, [5] := 2#0000_1011_0001_1101, [6] := 2#0000_1011_0001_1101, [7] := 2#0000_1011_0001_1101);
   O25_000 : ALIAS FOR O25[0];
   O25_001 : ALIAS FOR O25[1];
   O25_002 : ALIAS FOR O25[2];
   O25_003 : ALIAS FOR O25[3];
   O25_004 : ALIAS FOR O25[4];
   O25_005 : ALIAS FOR O25[5];
   O25_006 : ALIAS FOR O25[6];
   O25_007 : ALIAS FOR O25[7];
   O26 : INT[8] := ([0] := 2#0000_1010_0001_1101, [1] := 2#0000_1010_0001_1101, [2] := 2#0000_1010_0001_1101, [3] := 2#0000_1010_0001_1101, [4] := 2#0000_1010_0001_1101, [5] := 2#0000_1010_0001_1101, [6] := 2#0000_1010_0001_1101, [7] := 2#0000_1010_0001_1101);
   O26_000 : ALIAS FOR O26[0];
   O26_001 : ALIAS FOR O26[1];
   O26_002 : ALIAS FOR O26[2];
   O26_003 : ALIAS FOR O26[3];
   O26_004 : ALIAS FOR O26[4];
   O26_005 : ALIAS FOR O26[5];
   O26_006 : ALIAS FOR O26[6];
   O26_007 : ALIAS FOR O26[7];
   O27 : INT[4] := ([0] := 2#0110_0110_1001_1001, [1] := 2#0110_0110_1001_1001);
   O27_000 : ALIAS FOR O27[0];
   O27_001 : ALIAS FOR O27[1];
   O27_002 : ALIAS FOR O27[2];
   O27_003 : ALIAS FOR O27[3];
   O28 : INT[8] := ([0] := 2#0000_1011_0001_1101, [1] := 2#0000_1011_0001_1101, [2] := 2#0000_1011_0001_1101, [3] := 2#0000_0011_0000_1101);
   O28_000 : ALIAS FOR O28[0];
   O28_001 : ALIAS FOR O28[1];
   O28_002 : ALIAS FOR O28[2];
   O28_003 : ALIAS FOR O28[3];
   O28_004 : ALIAS FOR O28[4];
   O28_005 : ALIAS FOR O28[5];
   O28_006 : ALIAS FOR O28[6];
   O28_007 : ALIAS FOR O28[7];
   old_o13_3 : BOOL := 1;
   ONS1 : DINT;
   ons12 : BOOL;
   ONS13 : BOOL;
   onS14 : BOOL;
   onS15 : BOOL;
   onS16 : BOOL;
   ONS2 : BOOL;
   ONS3 : BOOL := 1;
   ONS4 : BOOL := 1;
   ONS5 : BOOL;
   ons6 : BOOL;
   ons7 : BOOL := 1;
   ons8 : BOOL := 1;
   ons9 : BOOL := 1;
   op010 : DINT := 439;
   P11_RECUP : BOOL := 1;
   P13_RECUP : BOOL := 1;
   P14_RECUP : BOOL;
   p15 : BOOL;
   P16 : BOOL := 1;
   P17 : BOOL;
   P18 : BOOL;
   P1_ETANG : BOOL := 1;
   P23 : BOOL;
   P24 : BOOL;
   P2_ETANG : BOOL;
   P3 : BOOL;
   P4 : BOOL := 1;
   P5_regen : BOOL;
   passage_jourmois : BOOL;
   pd3 : BOOL;
   pd4 : BOOL;
   pd5 : BOOL;
   pd6 : BOOL := 1;
   PD7 : BOOL;
   PD8 : BOOL := 1;
   PH11 : REAL := 57.63638;
   PH12 : REAL := -35.00267;
   PH2_PRETRAIT : REAL := 48.73274;
   PM1 : BOOL := 1;
   PM2 : BOOL := 1;
   PM3 : BOOL;
   PM4 : BOOL;
   PMP_L1_ET_L3_RUN : BOOL := 1;
   pmpput1 : BOOL := 1;
   pmpput2 : BOOL := 1;
   POS_EV3 : BOOL;
   PRES_LIGNE : REAL := 341.4969;
   Q2 : REAL := 87.743195;
   Q3 : REAL := 93.049515;
   Q4 : REAL := -38.681618;
   QUAT_Q1 : REAL := 170.0;
   QUAT_Q2 : REAL := 166.3363;
   R6 : CONTROL[1];
   real : REAL := 789.5018;
   S : INT[164] := ([0] := 16#0008, [1] := 16#00f6, [2] := 16#1032, [3] := 16#0c01, [4] := 16#b54e, [5] := 16#4000, [6] := 16#0021, [11] := 16#ffff, [12] := 16#ffff, [14] := 16#0032, [15] := 16#0b1b, [17] := 16#0002, [20] := 16#0002, [21] := 16#0002, [22] := 16#0006, [23] := 16#0005, [27] := 16#ffff, [28] := 16#ffff, [33] := 16#0008, [34] := 16#0002, [35] := 16#002f, [37] := 16#07e0, [38] := 16#000a, [39] := 16#0014, [40] := 16#000f, [41] := 16#0008, [42] := 16#0016, [53] := 16#0004, [57] := 16#0191, [58] := 16#0001, [59] := 16#0007, [60] := 16#021f, [61] := 16#0001, [62] := 16#0003, [63] := 16#0401, [64] := 16#0023, [65] := 16#0040, [66] := 16#0200, [83] := 16#0046, [84] := 16#f901, [85] := 16#0001, [86] := 16#01b1);
   S1 : BOOL;
   S24 : ALIAS FOR S[24];
   s_acide_ibt_passe : REAL := 26.200027;
   S_air_comp_Ecotech : REAL := 654.9172;
   S_AV310_V1_FC_C : BOOL := 1;
   S_AV310_V1_FC_O : BOOL;
   S_AV310_V2_FC_C : BOOL;
   S_AV310_V2_FC_O : BOOL := 1;
   S_AV320_V1_FC_C : BOOL := 1;
   S_AV320_V1_FC_O : BOOL;
   S_AV320_V2_FC_C : BOOL;
   S_AV320_V2_FC_O : BOOL := 1;
   S_AV330_V1_FC_C : BOOL;
   S_AV330_V1_FC_O : BOOL := 1;
   S_AV330_V2_FC_C : BOOL := 1;
   S_AV330_V2_FC_O : BOOL;
   S_BP_L2L3 : BOOL;
   s_bp_start_h2so4_ibt : BOOL;
   s_bp_stop_acide_ibt : BOOL;
   s_bp_stop_soude_ibt : BOOL;
   s_bp_wissel_P2_usi_tfb : BOOL;   // choix p2 etang vers tfb (1) ou usine (0)
   S_cond_Ecotech : REAL := 647.7455;
   S_COND_KOELTOREN : DINT := 3805;
   S_cond_venturi : DINT := -1000;
   S_def_airco_hT_l1 : BOOL;
   S_def_ventilo_hT_l1 : BOOL;
   s_dmd_acid_ibt : DINT := 150;
   S_dmd_naoh_ibt : REAL := 50.0;
   s_flow_lancy_L1 : REAL;
   s_flow_lancy_L2 : REAL := 44.63264;
   s_flow_lancy_L3 : REAL := 0.022888534;
   S_FLOW_PUT_1 : DINT := -30;
   S_FLOW_PUT_2 : DINT := -25;
   S_FLOW_VENTURI : DINT := 48;
   s_flw_filtrat_flt_presse : REAL := 165.55276;
   s_h2so4_ibt : BOOL;
   s_hac_turbidity : REAL := -250.01907;
   S_L2L3_Q_NAOH : DINT := 27;
   s_lastmonth_tot_h2o_l1 : REAL := 11528.477;
   s_lastmonth_tot_h2o_l2 : REAL := 11069.93;
   s_lastmonth_tot_h2o_l3 : REAL := 30721.078;
   s_lvl_apu_feed_TK : DINT := 789;
   s_lvl_buffert_flt_presse : REAL := 632.71533;
   s_lvl_filter_feed_TK : REAL := 511.9402;
   s_lvl_filtraat_water_from_flt : DINT := 269;
   s_lvl_holding_tk : REAL;
   S_Lvl_incident_bak : DINT := 12;
   S_LVL_KOELTOREN : DINT := 856;
   s_lvl_lift_tk : REAL := 525.3681;
   S_LVL_nitric : REAL := 1330.5867;
   s_lvl_op006 : REAL := 198.75258;
   s_lvl_op007 : REAL := 284.20007;
   s_lvl_op008 : REAL := 333.74;
   s_lvl_op009 : REAL := 762.1584;
   s_lvl_op010 : REAL := 437.77295;
   s_lvl_op011 : REAL := 309.77112;
   s_lvl_pellets_L4 : REAL := 61.570152;
   s_lvl_Ph_bac : REAL := -250.01907;
   s_lvl_puisard_L123 : REAL := 608.6824;
   s_lvl_reacteur_lancy : REAL := 889.0669;
   S_LVL_VIJVER : REAL := 72.480354;
   s_lvl_water_feed_TK : REAL := 808.423;
   S_naoh_ibt : BOOL;
   S_naoh_ibt_passe : REAL := 0.2;
   s_optek_turbidity : REAL := -250.01907;
   S_PH_naar_venturi : DINT := 775;
   S_Ph_Neutral : DINT := 794;
   S_PH_venturi : DINT := 701;
   s_pos_V_filtrat : REAL := -25.001907;
   S_pos_V_renv : DINT := 609;
   s_pos_V_venturi_open : BOOL := 1;
   S_ppas_HT : DINT := 5;
   S_ppas_l1op008 : DINT := 5;
   S_ppas_L2op008 : DINT := 5;
   S_STOCK_H2SO4 : DINT := 17654;
   S_STOCK_MAZ : DINT := 9202;
   S_STOCK_NAOH : DINT := 24829;
   S_stock_v_h2so4_f : BOOL := 1;
   S_stock_v_h2so4_o : BOOL;
   S_stock_v_naoh_f : BOOL := 1;
   S_stock_v_naoh_o : BOOL;
   S_T_CABINE_RED : DINT := 281;
   S_T_in_CH_L3 : DINT := 2135;
   S_T_in_chaud_L123 : DINT := -750;
   S_T_IWTS : DINT := 2184;
   S_T_OUT_CH_L3 : DINT := 2143;
   S_T_out_chaud_L123 : DINT := -750;
   S_T_venturi : DINT := -75;
   s_tot_vent_day : REAL := 954.0;
   s_V_h2so4 : BOOL;
   s_V_naoh : BOOL;
   scp_110 : SCP := (Input := 15684.0, Input_Min := 3277.0, Input_Max := 16384.0, Scaled_Max := 100.0, Output := 94.65934);
   Scp_air_comp_Ecotech : SCP := (Input := 11860.0, Input_Min := 3277.0, Input_Max := 16384.0, Scaled_Max := 1000.0, Output := 654.8409);
   scp_bas1 : SCP := (Input_Min := 3277.0, Input_Max := 16384.0, Scaled_Max := 300.0, Output := -75.00572);
   scp_cdro1 : SCP := (Input := 4260.0, Input_Min := 3277.0, Input_Max := 16384.0, Scaled_Max := 200.0, Output := 14.999619);
   scp_cdro2 : SCP := (Input := 3277.0, Input_Min := 3277.0, Input_Max := 16384.0, Scaled_Max := 200.0);
   scp_cdro3 : SCP := (Input := 16384.0, Input_Min := 3277.0, Input_Max := 16384.0, Scaled_Max := 200.0, Output := 200.0);
   scp_COND1 : SCP := (Input_Min := 3277.0, Input_Max := 16384.0, Scaled_Max := 5000.0, Output := -1250.0953);
   scp_COND2_OS : SCP := (Input := 1267.0, Input_Min := 3277.0, Input_Max := 16384.0, Scaled_Max := 2000.0, Output := -306.70633);
   scp_COND3 : SCP := (Input := 1749.0, Input_Max := 10000.0, Scaled_Max := 2000.0, Output := 349.80002);
   scp_COND4 : SCP := (Input := 2552.0, Input_Max := 10000.0, Scaled_Max := 1000.0, Output := 255.2);
   scp_COND7 : SCP := (Input_Min := 3277.0, Input_Max := 16384.0, Scaled_Min := 40.0, Scaled_Max := 200.0, Output := -0.0030517578);
   Scp_cond_Ecotech : SCP := (Input := 6113.0, Input_Min := 3277.0, Input_Max := 16384.0, Scaled_Max := 3000.0, Output := 649.1188);
   SCP_COND_KOELTOREN : SCP := (Input := 7852.0, Input_Min := 3277.0, Input_Max := 16383.0, Scaled_Max := 10000.0, Output := 3490.7676);
   scp_cond_venturi : SCP := (Input_Min := 3277.0, Input_Max := 16383.0, Scaled_Min := 20.0, Scaled_Max := 3000.0, Output := -725.1137);
   scp_EAU_VILLE : SCP := (Input_Min := 3277.0, Input_Max := 16384.0, Scaled_Max := 140.0, Output := -35.00267);
   scp_flow_lancy_L1 : SCP := (Input := 3277.0, Input_Min := 3277.0, Input_Max := 16384.0, Scaled_Max := 100.0);
   scp_flow_lancy_L2 : SCP := (Input := 9116.0, Input_Min := 3277.0, Input_Max := 16384.0, Scaled_Max := 100.0, Output := 44.548714);
   scp_flow_lancy_L3 : SCP := (Input := 3281.0, Input_Min := 3277.0, Input_Max := 16384.0, Scaled_Max := 100.0, Output := 0.030518044);
   scp_flvl_op006 : SCP := (Input := 7377.0, Input_Min := 3277.0, Input_Max := 16384.0, Scaled_Min := 30.0, Scaled_Max := 570.0, Output := 198.91737);
   scp_flvl_op007 : SCP := (Input := 9445.0, Input_Min := 3277.0, Input_Max := 16384.0, Scaled_Min := 30.0, Scaled_Max := 570.0, Output := 284.11765);
   scp_flvl_op008 : SCP := (Input := 6284.0, Input_Min := 3277.0, Input_Max := 16384.0, Scaled_Min := 30.0, Scaled_Max := 1350.0, Output := 332.8336);
   scp_flvl_op009 : SCP := (Input := 10548.0, Input_Min := 3277.0, Input_Max := 16384.0, Scaled_Min := 30.0, Scaled_Max := 1350.0, Output := 762.2591);
   scp_flvl_op010 : SCP := (Input := 7326.0, Input_Min := 3277.0, Input_Max := 16384.0, Scaled_Min := 30.0, Scaled_Max := 1350.0, Output := 437.77295);
   scp_flvl_op011 : SCP := (Input := 6061.0, Input_Min := 3277.0, Input_Max := 16384.0, Scaled_Min := 30.0, Scaled_Max := 1350.0, Output := 310.37537);
   scp_FLW_CO1 : SCP := (Input := 6103.0, Input_Min := 3277.0, Input_Max := 16384.0, Scaled_Max := 200.0, Output := 43.121994);
   scp_FLW_CO2 : SCP := (Input := 3277.0, Input_Min := 3277.0, Input_Max := 16384.0, Scaled_Max := 200.0);
   scp_FLW_CO3 : SCP := (Input := 3279.0, Input_Min := 3277.0, Input_Max := 16384.0, Scaled_Max := 200.0, Output := 0.030518044);
   scp_flw_filtrat_flt_presse : SCP := (Input := 8097.0, Input_Min := 3277.0, Input_Max := 16384.0, Scaled_Max := 450.0, Output := 165.4841);
   scp_FLW_PO1 : SCP := (Input := 10217.0, Input_Min := 3277.0, Input_Max := 16384.0, Scaled_Max := 300.0, Output := 158.84642);
   scp_FLW_PO2 : SCP := (Input := 3277.0, Input_Min := 3277.0, Input_Max := 16384.0, Scaled_Max := 300.0);
   scp_FLW_PO3 : SCP := (Input := 3281.0, Input_Min := 3277.0, Input_Max := 16384.0, Scaled_Max := 300.0, Output := 0.091554135);
   scp_flw_put1 : SCP := (Input_Min := 3277.0, Input_Max := 16383.0, Scaled_Max := 100.0, Output := -25.003815);
   scp_flw_put2 : SCP := (Input_Min := 3277.0, Input_Max := 16383.0, Scaled_Max := 100.0, Output := -25.003815);
   scp_flw_put3 : SCP := (Input_Min := 3277.0, Input_Max := 16383.0, Scaled_Max := 120.0, Output := -30.004578);
   scp_FLW_Q3 : SCP := (Input := 9352.0, Input_Min := 3277.0, Input_Max := 16384.0, Scaled_Max := 200.0, Output := 92.698555);
   scp_flw_venturi : SCP := (Input_Min := 3277.0, Input_Max := 16383.0, Scaled_Max := 180.0, Output := -45.006866);
   scp_hac_turbidity : SCP := (Input_Min := 3277.0, Input_Max := 16384.0, Scaled_Max := 1000.0, Output := -250.01907);
   scp_hard : SCP := (Input_Min := 3277.0, Input_Max := 16384.0, Scaled_Max := 100.0, Output := -25.001907);
   scp_KR_1 : SCP := (Input := 16024.0, Input_Min := 3277.0, Input_Max := 16384.0, Scaled_Min := 550.0, Scaled_Max := 206.0, Output := 215.4484);
   scp_KRK2 : SCP := (Input := 12234.0, Input_Min := 3277.0, Input_Max := 16384.0, Scaled_Min := 440.0, Scaled_Max := 230.0, Output := 296.4912);
   scp_l1_flow : SCP := (Input := 4747.0, Input_Max := 10000.0, Scaled_Max := 500.0, Output := 237.35);
   scp_l2_flow : SCP := (Input := 4854.0, Input_Max := 10000.0, Scaled_Max := 500.0, Output := 242.7);
   scp_l3_flow : SCP := (Input := 4848.0, Input_Max := 10000.0, Scaled_Max := 500.0, Output := 242.40001);
   scp_LDN_1 : SCP := (Input := 3781.0, Input_Min := 3277.0, Input_Max := 16384.0, Scaled_Min := 340.0, Scaled_Max := 140.0, Output := 332.30945);
   scp_LDN_2 : SCP := (Input := 14742.0, Input_Min := 3277.0, Input_Max := 16384.0, Scaled_Min := 340.0, Scaled_Max := 140.0, Output := 165.05531);
   scp_LDN_3 : SCP := (Input := 13646.0, Input_Min := 3277.0, Input_Max := 16384.0, Scaled_Min := 400.0, Scaled_Max := 200.0, Output := 241.7792);
   scp_LUS2 : SCP := (Input := 14268.0, Input_Min := 3277.0, Input_Max := 16384.0, Scaled_Max := 1000.0, Output := 838.5595);
   scp_LUS3 : SCP := (Input := 14167.0, Input_Min := 3277.0, Input_Max := 16384.0, Scaled_Max := 1000.0, Output := 830.8537);
   scp_lvl_apu_feed_TK : SCP := (Input := 13625.0, Input_Min := 3277.0, Input_Max := 16384.0, Scaled_Max := 1000.0, Output := 789.5018);
   scp_LVL_AZ : SCP := (Input := 7884.0, Input_Max := 10000.0, Scaled_Max := 100.0, Output := 78.84);
   scp_lvl_buffer_flt_presse : SCP := (Input := 11563.0, Input_Min := 3277.0, Input_Max := 16384.0, Scaled_Max := 1000.0, Output := 632.1813);
   scp_lvl_filter_feed_TK : SCP := (Input := 9987.0, Input_Min := 3277.0, Input_Max := 16384.0, Scaled_Max := 1000.0, Output := 511.9402);
   scp_lvl_filtraat_water_from_flt : SCP := (Input := 10327.0, Input_Min := 3277.0, Input_Max := 16384.0, Scaled_Max := 500.0, Output := 268.94025);
   scp_lvl_holding_tk : SCP := (Input := 3277.0, Input_Min := 3277.0, Input_Max := 16384.0, Scaled_Max := 1000.0);
   SCP_LVL_KOELTOREN : SCP := (Input := 14524.0, Input_Min := 3277.0, Input_Max := 16384.0, Scaled_Max := 1000.0, Output := 858.09106);
   scp_lvl_l4 : SCP := (Input_Min := 3277.0, Input_Max := 16383.0, Scaled_Max := 100.0, Output := -25.003815);
   scp_lvl_lift_tk : SCP := (Input := 10152.0, Input_Min := 3277.0, Input_Max := 16384.0, Scaled_Max := 1000.0, Output := 524.5289);
   SCP_lvl_nitric : SCP := (Input := 6759.0, Input_Min := 3277.0, Input_Max := 16384.0, Scaled_Max := 5000.0, Output := 1328.2979);
   scp_lvl_pellets_L4 : SCP := (Input := 4083.0, Input_Min := 3277.0, Input_Max := 16384.0, Scaled_Max := 1000.0, Output := 61.49386);
   scp_lvl_Ph_bac : SCP := (Input_Min := 3277.0, Input_Max := 16384.0, Scaled_Max := 1000.0, Output := -250.01907);
   scp_LVL_PRET : SCP := (Input := 14313.0, Input_Min := 3277.0, Input_Max := 16384.0, Scaled_Max := 100.0, Output := 84.19928);
   scp_LVL_PUIS : SCP := (Input := 6580.0, Input_Min := 3277.0, Input_Max := 16384.0, Scaled_Max := 1000.0, Output := 252.00275);
   scp_LVL_PUIS_L4 : SCP := (Input_Min := 3277.0, Input_Max := 16384.0, Scaled_Max := 100.0, Output := -25.001907);
   scp_lvl_puisard_L123 : SCP := (Input := 11258.0, Input_Min := 3277.0, Input_Max := 16384.0, Scaled_Max := 1000.0, Output := 608.91125);
   scp_lvl_reacteur_lancy : SCP := (Input := 14920.0, Input_Min := 3277.0, Input_Max := 16384.0, Scaled_Max := 1000.0, Output := 888.30396);
   scp_lvl_vijver : SCP := (Input := 12785.0, Input_Min := 3277.0, Input_Max := 16384.0, Scaled_Max := 100.0, Output := 72.54139);
   scp_lvl_water_feed_TK : SCP := (Input := 13873.0, Input_Min := 3277.0, Input_Max := 16384.0, Scaled_Max := 1000.0, Output := 808.423);
   scp_LVL_ZOUT : SCP := (Input_Min := 3277.0, Input_Max := 16384.0, Scaled_Max := 100.0, Output := -25.001907);
   scp_N12_14 : SCP := (Input := 5996.0, Input_Max := 10000.0, Scaled_Max := 150.0, Output := 89.939995);
   scp_N12_219 : SCP := (Input := 16384.0, Input_Min := 3277.0, Input_Max := 16384.0, Scaled_Max := 1000.0, Output := 1000.0);
   scp_N12_220 : SCP := (Input := 8487.0, Input_Min := 3277.0, Input_Max := 16384.0, Scaled_Max := 1000.0, Output := 397.4975);
   scp_N12_221 : SCP := (Input_Min := 3277.0, Input_Max := 16384.0, Scaled_Max := 1000.0, Output := -250.01907);
   scp_N12_38 : SCP := (Input := 4998.0, Input_Max := 10000.0, Scaled_Max := 2000.0, Output := 999.60004);
   scp_N12_44 : SCP := (Input := -2501.0, Input_Max := 10000.0, Scaled_Max := 2000.0, Output := -500.2);
   scp_N7_70 : SCP := (Input := 8046.0, Input_Max := 10000.0, Scaled_Max := 100.0, Output := 80.46);
   scp_N7_71 : SCP := (Input := 9904.0, Input_Max := 10000.0, Scaled_Max := 100.0, Output := 99.04);
   scp_N7_72 : SCP := (Input := 7824.0, Input_Max := 10000.0, Scaled_Max := 2000.0, Output := 1564.8);
   scp_optek_turbidity : SCP := (Input_Min := 3277.0, Input_Max := 16384.0, Scaled_Max := 1000.0, Output := -250.01907);
   scp_PH11 : SCP := (Input := 8209.0, Input_Min := 3277.0, Input_Max := 16384.0, Scaled_Min := 20.0, Scaled_Max := 120.0, Output := 57.62875);
   scp_PH12 : SCP := (Input_Min := 3277.0, Input_Max := 16384.0, Scaled_Max := 140.0, Output := -35.00267);
   scp_PH2 : SCP := (Input := 7046.0, Input_Min := 3277.0, Input_Max := 16384.0, Scaled_Min := 20.0, Scaled_Max := 120.0, Output := 48.755627);
   scp_ph_venturi : SCP := (Input_Min := 3277.0, Input_Max := 16383.0, Scaled_Max := 140.0, Output := -35.00534);
   scp_pos_V_filtrat : SCP := (Input_Min := 3277.0, Input_Max := 16384.0, Scaled_Max := 100.0, Output := -25.001907);
   scp_PRES_LIGNE : SCP := (Input := 7747.0, Input_Min := 3277.0, Input_Max := 16384.0, Scaled_Max := 1000.0, Output := 341.03912);
   scp_Q2 : SCP := (Input := 10960.0, Input_Min := 3277.0, Input_Max := 16384.0, Scaled_Max := 150.0, Output := 87.9263);
   scp_Q4 : SCP := (Input := 2796.0, Input_Min := 3277.0, Input_Max := 16384.0, Scaled_Max := 1000.0, Output := -36.69795);
   scp_quat_2 : SCP := (Input := 3781.0, Input_Min := 3277.0, Input_Max := 16384.0, Scaled_Min := 170.0, Scaled_Max := 72.0, Output := 166.23163);
   scp_QUAT_Q1 : SCP := (Input := 3277.0, Input_Min := 3277.0, Input_Max := 16384.0, Scaled_Min := 170.0, Scaled_Max := 140.0, Output := 170.0);
   SCP_SPEED_PMP_FAB : SCP := (Input := 75.20038, Input_Max := 100.0, Scaled_Min := 6550.0, Scaled_Max := 32767.0, Output := 26265.285);
   scp_stck_acid : SCP := (Input := 12498.0, Input_Min := 3277.0, Input_Max := 16383.0, Scaled_Max := 25092.0, Output := 17654.0);
   scp_stck_maz : SCP := (Input := 5688.0, Input_Min := 3277.0, Input_Max := 16383.0, Scaled_Max := 50000.0, Output := 9198.077);
   scp_stck_soude : SCP := (Input := 9918.0, Input_Min := 3277.0, Input_Max := 16383.0, Scaled_Max := 49000.0, Output := 24829.01);
   SCP_T_CABINE_L1 : SCP := (Input := 6966.0, Input_Min := 3277.0, Input_Max := 16384.0, Scaled_Max := 1000.0, Output := 281.45264);
   scp_T_in_CH_L3 : SCP := (Input := 12605.0, Input_Min := 3277.0, Input_Max := 16383.0, Scaled_Max := 3000.0, Output := 2135.205);
   scp_T_in_L12 : SCP := (Input_Min := 3277.0, Input_Max := 16383.0, Scaled_Max := 3000.0, Output := -750.11444);
   scp_T_iwts : SCP := (Input := 12832.0, Input_Min := 3277.0, Input_Max := 16383.0, Scaled_Max := 3000.0, Output := 2187.166);
   scp_T_OUT_CH_L3 : SCP := (Input := 12638.0, Input_Min := 3277.0, Input_Max := 16383.0, Scaled_Max := 3000.0, Output := 2142.759);
   scp_T_out_L12 : SCP := (Input_Min := 3277.0, Input_Max := 16383.0, Scaled_Max := 3000.0, Output := -750.11444);
   scp_t_venturi : SCP := (Input_Min := 3277.0, Input_Max := 16383.0, Scaled_Max := 100.0, Output := -25.003815);
   scpcond_6 : SCP := (Input_Min := 3277.0, Input_Max := 16383.0, Scaled_Max := 1958.0, Output := -489.5747);
   Seconde : BOOL := 1;
   soude_ibt_fini : BOOL := 1;
   SPEED_P3 : DINT := 26265;
   stat_L1 : DINT[20] := ([1] := 589824, [3] := 50, [4] := 2, [5] := 888, [19] := 20); {produced}
        [13].6   // demande nitrique
        [13].0   // run nitrique vers L1
        [1].0   // fuite acide au stock
        [1].1   // fuite soude au stock
        [1].2   // fuite mazout au stock
        [1].4   // de plc stock apport soude finit
        [1].12   // DEFAULT NaOH fill up
        [1].6   // de plc stock apport soude accordé
        [1].5   // de plc stock apport soude occupé
        [1].7   // de plc stock soude vers l1
        [1].8   // de plc stock soude vers L2
        [1].9   // de plc stock soude vers L3
        [1].10   // de plc stock soude vers L4
        [1].11   // de plc stock soude vers stat
        [1].3   // de plc stock ouverture vanne soude
        [2].4   // apport acide finit
        [0]   // de plc stock soude restante
        [2].3   // ouvrir vanne acide
        [2].5   // apport acide occupé
        [2].6   // apport acide accordé
        [2].7   // acide vers l1
        [2].8   // acide vers l2
        [2].9   // acide vers l3
        [2].10   // acide vers l4
        [2].11   // acide vers neut L1
        [2].12   // acide vers neut L2
        [2].13   // acide vers neut L3
        [2].14   // acide vers neut L4
        [2].15   // quantite acide passé
   STAT_L2 : DINT[20] := ([1] := 393216, [3] := 300, [4] := 2, [5] := 888, [6] := 45); {produced}
        [13].6   // demande nitrique
        [13].0   // run nitrique vers L2
        [0]   // de plc stock soude restante
        [1].3   // de plc stock ouverture vanne soude
        [1].4   // de plc stock apport soude finit
        [1].5   // de plc stock apport soude occupé
        [1].6   // de plc stock apport soude accordé
        [1].7   // de plc stock soude vers l1
        [1].8   // de plc stock soude vers L2
        [1].9   // de plc stock soude vers L3
        [1].10   // de plc stock soude vers L4
        [1].11   // de plc stock soude vers STAT
        [1].12   // DEFAULT NaOH fill up
        [2].3   // ouvrir vanne acide
        [2].4   // apport acide finit
        [2].5   // apport acide occupé
        [2].6   // apport acide accordé
        [2].7   // acide vers l1
        [2].8   // acide vers l2
        [2].9   // acide vers l3
        [2].10   // acide vers l4
        [2].11   // acide vers neut L1
        [2].12   // acide vers neut L2
        [2].13   // acide vers neut L3
        [2].14   // acide vers neut L4
        [2].15   // quantite acide passé
   STAT_L3 : DINT[20] := ([1] := 393216, [3] := 200, [4] := 2, [5] := 888, [12] := 143130); {produced}
        [13].6   // demande nitrique
        [13].0   // run nitrique vers L3
        [0]   // de plc stock soude restante
        [1].0   // REQGRSDQ
        [1].3   // de plc stock ouverture vanne soude
        [1].4   // de plc stock apport soude finit
        [1].5   // de plc stock apport soude occupé
        [1].6   // de plc stock apport soude accordé
        [1].7   // de plc stock soude vers l1
        [1].8   // de plc stock soude vers L2
        [1].9   // de plc stock soude vers L3
        [1].10   // de plc stock soude vers L4
        [1].11   // de plc stock soude vers STAT
        [1].12   // DEFAULT NaOH fill up
        [2].3   // ouvrir vanne acide
        [2].4   // apport acide finit
        [2].5   // apport acide occupé
        [2].6   // apport acide accordé
        [2].7   // acide vers l1
        [2].8   // acide vers l2
        [2].9   // acide vers l3
        [2].10   // acide vers l4
        [2].11   // acide vers neut L1
        [2].12   // acide vers neut L2
        [2].13   // acide vers neut L3
        [2].14   // acide vers neut L4
        [2].15   // quantite acide passé
   STAT_wkk : DINT[20]; {produced}
   Status : INT := 12640;   // INT tag to retrieve Status value through GSV created during conversion
   STEP_DUALM_3_4_5_6 : BOOL;
   STEP_NASPOEL_1_ET_2 : BOOL := 1;
   STEP_REI_Z_2_3_6_7 : BOOL;
   STEP_REI_Z_2_3_6_7B : BOOL;
   STEP_REO_Z_2_6_A_ET_B : BOOL;
   stocklancy1 : DINT := 91;
   stocklancy2 : DINT;
   stocklancy3 : DINT := 10;
        .0   // NAOHL1 VA4FC O
        .1   // NAOHL1 VA4FC F
        .2   // NAOHL2 VA4FC O
        .3   // NAOHL2 VA4FC O
   stocklancy4 : DINT := 7;   // alarme lvl 1 stock
   stocklancy5 : DINT := 3;   // alarme lvl 2 stock
   t1 : TIMER := (PRE := 30000);
   T1_cligno : TIMER := (PRE := 500, ACC := 50, EN := 1, TT := 1);
   t1min : TIMER := (PRE := 60000, ACC := 47050, EN := 1, TT := 1);
   t1sec : TIMER := (PRE := 1100, ACC := 750, EN := 1, TT := 1);
   T27 : TIMER[100] := ([0].PRE := 15000, [0].ACC := 15000, [0].EN := 1, [0].DN := 1, [1].PRE := 15000, [2].PRE := 15000, [3].PRE := 50, [3].ACC := 50, [3].EN := 1, [3].DN := 1, [4].PRE := 50, [4].ACC := 50, [4].EN := 1, [4].DN := 1, [5].PRE := 50, [5].ACC := 50, [5].EN := 1, [5].DN := 1, [6].PRE := 6000000, [6].ACC := 5441400, [6].EN := 1, [6].TT := 1, [7].PRE := 60000, [10].PRE := 32000000, [10].ACC := 32000000, [10].EN := 1, [10].DN := 1, [11].PRE := 32000000, [11].ACC := 31128400, [11].EN := 1, [11].TT := 1, [12].PRE := 10000, [12].ACC := 6600, [12].EN := 1, [12].TT := 1, [13].PRE := 10000, [14].PRE := 500, [14].ACC := 520, [14].EN := 1, [14].DN := 1, [15].PRE := 500, [15].ACC := 340, [15].EN := 1, [15].TT := 1, [16].PRE := 5000, [17].PRE := 5000, [18].PRE := 5000, [19].PRE := 500, [19].ACC := 500, [19].EN := 1, [19].DN := 1, [20].PRE := 10000, [21].PRE := 5000, [21].ACC := 5000, [21].EN := 1, [21].DN := 1, [22].PRE := 3000, [22].ACC := 3000, [23].PRE := 3000, [23].ACC := 3000,
        [24].PRE := 50, [24].ACC := 50, [24].EN := 1, [24].DN := 1, [25].PRE := 10, [25].ACC := 50, [25].EN := 1, [25].DN := 1, [26].PRE := 3600000, [26].ACC := 1694800, [26].EN := 1, [26].TT := 1, [27].PRE := 5000, [27].ACC := 5049, [27].EN := 1, [27].DN := 1, [29].PRE := 10000, [29].ACC := 10000, [40].PRE := 120000, [41].PRE := 120000, [42].PRE := 120000, [47].PRE := 50, [47].ACC := 50, [47].EN := 1, [47].DN := 1, [48].PRE := 50, [48].ACC := 50, [48].EN := 1, [48].DN := 1, [49].PRE := 50, [49].ACC := 50, [49].EN := 1, [49].DN := 1, [50].PRE := 5000, [50].ACC := 5000, [50].EN := 1, [50].DN := 1, [51].PRE := 960000, [52].PRE := 60000, [53].PRE := 5000, [54].PRE := 900000, [55].PRE := 60000, [56].PRE := 5000, [57].PRE := 960000, [58].PRE := 60000, [59].PRE := 10000, [59].ACC := 10000, [59].EN := 1, [59].DN := 1, [60].PRE := 1000, [60].ACC := 1000, [60].EN := 1, [60].DN := 1, [62].PRE := 5000, [63].PRE := 50, [63].ACC := 50, [63].EN := 1, [63].DN := 1, [65].PRE := 5000, [66].PRE := 50,
        [66].ACC := 50, [66].EN := 1, [66].DN := 1, [67].PRE := 15000, [67].ACC := 15000, [67].EN := 1, [67].DN := 1, [68].PRE := 15000, [69].PRE := 15000, [70].PRE := 900000, [71].PRE := 600000, [72].PRE := 600000, [75].PRE := 7200000, [75].ACC := 7200000, [76].PRE := 7200000, [76].ACC := 7200000, [77].PRE := 5000, [78].PRE := 5000, [79].PRE := 5, [80].PRE := 3600000, [80].EN := 1, [80].DN := 1, [81].ACC := 50, [81].EN := 1, [81].DN := 1, [82].PRE := 500000, [82].ACC := 391050, [82].EN := 1, [82].TT := 1, [83].PRE := 5000, [84].PRE := 5000, [87].PRE := 100, [87].ACC := 100, [87].EN := 1, [87].DN := 1, [88].PRE := 100, [88].ACC := 36, [88].EN := 1, [88].TT := 1, [89].PRE := 120000, [89].ACC := 120000, [89].EN := 1, [89].DN := 1, [90].PRE := 120000, [90].ACC := 120000, [90].EN := 1, [90].DN := 1, [91].EN := 1, [91].DN := 1, [92].PRE := 3600, [92].ACC := 2012, [92].EN := 1, [92].TT := 1, [93].PRE := 10000, [94].PRE := 10000, [96].PRE := 10000);
   T2_cligno : TIMER := (PRE := 500);
   T4 : TIMER[200] := ([0].PRE := 200, [1].PRE := 120000, [1].ACC := 120000, [1].EN := 1, [1].DN := 1, [2].PRE := 120000, [2].ACC := 120000, [3].PRE := 5000, [3].ACC := 5000, [3].EN := 1, [3].DN := 1, [4].PRE := 1800000, [5].PRE := 300000, [6].PRE := 1800000, [6].ACC := 1800000, [6].EN := 1, [6].DN := 1, [7].PRE := 600000, [7].ACC := 600000, [8].PRE := 120000, [9].PRE := 120000, [9].ACC := 120000, [9].EN := 1, [9].DN := 1, [10].PRE := 300000, [11].PRE := 20000, [12].PRE := 900000, [13].PRE := 90000, [13].ACC := 90000, [14].PRE := 150000, [15].PRE := 5000, [16].PRE := 100000, [16].ACC := 3300, [16].TT := 1, [16].DN := 1, [17].PRE := 30000, [17].EN := 1, [17].DN := 1, [18].PRE := 5000, [18].ACC := 5000, [18].EN := 1, [18].DN := 1, [19].PRE := 5000, [19].ACC := 5000, [20].PRE := 7000, [21].PRE := 10000, [22].PRE := 300000, [23].PRE := 900000, [24].PRE := 20000, [25].PRE := 850000, [26].PRE := 60000, [27].PRE := 30000, [28].PRE := 5000, [29].PRE := 5000, [29].ACC := 5000, [29].EN := 1, [29].DN := 1, [30].PRE := 7000, [31].PRE := 10000, [32].PRE := 300000,
        [33].PRE := 900000, [34].PRE := 20000, [35].PRE := 850000, [36].PRE := 60000, [37].PRE := 30000, [38].PRE := 7000, [38].ACC := 7000, [38].EN := 1, [38].DN := 1, [39].PRE := 30000, [40].PRE := 15000, [41].PRE := 10000, [42].PRE := 30000, [43].PRE := 1200000, [44].PRE := 1800000, [45].PRE := 4500000, [46].PRE := 33000, [47].PRE := 10000, [47].ACC := 10000, [47].EN := 1, [47].DN := 1, [48].PRE := 30000, [48].EN := 1, [48].DN := 1, [49].PRE := 10000, [50].PRE := 15000, [51].PRE := 7000, [52].PRE := 30000, [53].PRE := 900000, [54].PRE := 1800000, [55].PRE := 4500000, [55].ACC := 1765450, [55].EN := 1, [55].TT := 1, [56].PRE := 33000, [57].PRE := 900000, [57].ACC := 900000, [58].PRE := 300000, [58].ACC := 300000, [60].PRE := 20000, [61].PRE := 60000, [62].PRE := 60000, [63].PRE := 30000, [64].PRE := 120000, [65].PRE := 700000, [66].PRE := 20000, [67].PRE := 850000, [68].PRE := 60000, [69].PRE := 60000, [70].PRE := 225, [71].PRE := 35000, [72].PRE := 10000, [73].PRE := 900000, [74].PRE := 1800000, [75].PRE := 4500000, [76].PRE := 35000, [76].ACC := 35000, [76].EN := 1, [76].DN := 1, [77].PRE := 1800000,
        [77].ACC := 1313400, [77].EN := 1, [77].TT := 1, [78].PRE := 14400000, [78].ACC := 14400000, [79].PRE := 300000, [79].ACC := 300049, [79].EN := 1, [79].DN := 1, [80].PRE := 15000, [81].PRE := 35000, [82].PRE := 10000, [83].PRE := 900000, [84].PRE := 1800000, [85].PRE := 4500000, [86].PRE := 35000, [87].PRE := 10000, [87].EN := 1, [87].DN := 1, [88].PRE := 300000, [90].PRE := 10000, [91].PRE := 50000, [92].PRE := 10000, [92].ACC := 10000, [92].EN := 1, [92].DN := 1, [93].PRE := 60000, [94].PRE := 120000, [94].ACC := 120000, [95].PRE := 1000, [95].ACC := 400, [95].EN := 1, [95].TT := 1, [96].PRE := 500, [97].PRE := 60000, [97].ACC := 47850, [97].EN := 1, [97].TT := 1, [98].PRE := 120000, [100].PRE := 10000, [101].PRE := 50000, [102].PRE := 10000, [103].PRE := 60000, [104].PRE := 300000, [105].PRE := 5000, [105].ACC := 2600, [105].EN := 1, [105].TT := 1, [106].PRE := 60000, [106].ACC := 60000, [106].EN := 1, [106].DN := 1, [107].PRE := 1000, [107].ACC := 650, [107].EN := 1, [107].TT := 1, [108].PRE := 1000, [110].PRE := 10000, [111].PRE := 50000, [112].PRE := 10000,
        [113].PRE := 60000, [114].PRE := 300000, [114].ACC := 300049, [114].EN := 1, [114].DN := 1, [120].PRE := 10000, [121].PRE := 1000, [122].PRE := 1000, [123].PRE := 9000000, [124].PRE := 6000000, [125].PRE := 1000, [126].PRE := 1000, [127].PRE := 1800000, [128].PRE := 600000, [129].PRE := 120000, [129].ACC := 120000, [130].PRE := 20000, [131].PRE := 1000, [132].PRE := 1000, [133].PRE := 18000000, [134].PRE := 600000, [135].PRE := 1000, [136].PRE := 1000, [137].PRE := 1800000, [138].PRE := 600000, [140].PRE := 5000, [141].PRE := 1000, [142].PRE := 1000, [143].PRE := 1800000, [144].PRE := 600000, [145].PRE := 1000, [146].PRE := 1000, [147].PRE := 1800000, [148].PRE := 1000, [149].PRE := 2000000, [150].PRE := 600000, [151].PRE := 1000, [152].PRE := 1000, [153].PRE := 1800000, [154].PRE := 600000, [155].PRE := 60000, [160].PRE := 30000, [161].PRE := 10000, [162].PRE := 10000, [163].PRE := 60000, [166].PRE := 30000, [167].PRE := 15000, [168].PRE := 15000, [169].PRE := 60000, [170].PRE := 80000, [170].ACC := 80000, [170].EN := 1, [170].DN := 1, [171].PRE := 60000, [171].ACC := 53700, [171].EN := 1, [171].TT := 1, [172].PRE := 60000, [172].ACC := 37250, [173].PRE := 60000,
        [173].ACC := 35950, [174].PRE := 60000, [174].ACC := 35500, [174].EN := 1, [174].TT := 1, [175].PRE := 60000, [175].ACC := 40250, [175].EN := 1, [175].TT := 1, [176].PRE := 60000, [176].ACC := 46050, [176].EN := 1, [176].TT := 1, [177].PRE := 60000, [177].ACC := 21950, [180].PRE := 600000, [180].ACC := 240050, [180].EN := 1, [180].TT := 1, [181].PRE := 300000, [181].ACC := 287350, [181].EN := 1, [181].TT := 1, [182].PRE := 900000, [182].ACC := 386850, [182].EN := 1, [182].TT := 1);
        [1]   // tempo niveau kuip 20m laag niv
        [2]   // laag alarm ketel tampon
        [3]   // tempo marche pompe puit 2
        [5]   // tempo start P24 by Ventury
        [7]   // tempo niveau kuip 20m hoog alarm
        [8]   // tempo attente redéarrage pmp puits
        [9]   // tempo attente redéarrage pmp étang
        [11]   // tempo niveau NACL
        [12]   // ?
        [13]   // ?
        [14]   // tempo pompe 1 puisard ligne 4
        [15]   // tempo pompe 2 puisard ligne 4
        [16]   // ?
        [17]   // ?
        [18]   // tempo marche pompe puit 3
        [19]   // tempo demande marche pmp puits
        [28]   // tempo defaut vanne pmp puits 2
        [29]   // tempo defaut vanne pmp puits 3
        [35]   // temps ajout d'eau rinçage
        [38]   // TEMPO POMPE OSMOSE MARCHE
        [39]   // TEMPO defaut VANNE ALIBERT
        [77]   // rappel si pas de réponse
        [78]   // acquit t
        [79]   // defaut PH venturi attent si pas un pic
        [95]   // tempo seconde
        [96]   // ?
        [97]   // T4:97
        [105]   // tempo envoi messagevers lancy
        [155]   // defaut vanne position eau ville
        [170]   // openning (osr) stfa1 ev1 ou stfa1 ev2 depuis + de 80 sec
        [171]   // tempo marche pmp 1 min
        [172]   // tempo marche pmp 1 min
        [173]   // tempo marche pmp 1 min
        [180]   // temps attente verif flow Q1
        [181]   // TEMPO CHECK EMPTYING TANK
        [182]   // temps attente verif flow Q2
   T_CABINE_RED : REAL := 281.22375;
   T_R_L2L3 : TIMER := (PRE := 90000);
   tempo_d_lvl_H_decL1 : TIMER := (PRE := 30000, ACC := 30000, EN := 1, DN := 1);
   tempo_on_lvl_H_decL1 : TIMER := (PRE := 30000);
   toff_def_flow : TIMER := (PRE := 3000, ACC := 3000);
   ton_run_eco : TIMER := (PRE := 30000);
   tot_gaz_chaud_iwts_L123 : DINT := 1483608;   // 19/1/15 13h45
   tot_gaz_chaud_L3 : DINT := 500876;   // debut le 16/1/15 à 11h30
   tot_gaz_chaud_wanson : DINT := 295214;   // 19/1/15 13h45
   tot_h2so4_stat : REAL;
   tot_pulse_venturi : REAL := 5745812.0;
   tot_put_1 : DINT := 66985;
   tot_put_2 : DINT := 180668;
   vanne_filtraaT : REAL := 19848.469;
   water_flow_to_l1 : REAL := 139764.12;
   water_flow_to_l1_inst : REAL := 38.4375;
   water_flow_to_l2 : REAL := 90148.34;
   water_flow_to_l2_inst : REAL := 20.625;
   water_flow_to_l3 : REAL := 205436.58;
   water_flow_to_l3_inst : DINT := 306;
   water_flow_to_l3_inst1 : REAL := 38.4375;
   wkk_STAT : DINT[20];
END_VAR

PROGRAM BASSIN   (* main routine main_Bassin *)
VAR
   B3 : DINT[10] := ([1] := 14);
        [1].3   // en cours augmentation PH
        [1].8   // ajout acide
        [2].0   // mauvais PH vers venturi
        [1].7   // ajout soude
   F8 : REAL[50] := ([1] := 428484.34, [2] := 792.5078, [3] := 429276.84, [4] := 793.4877, [5] := 0.81666666, [6] := 386178.22);
   N20 : DINT[50] := ([6] := 775, [7] := 701, [8] := 793, [11] := 841, [13] := 778, [15] := 783);
        [1]   // DEFAUT PRIORITE 1
        [2]   // DEFAUT PRIORITE 2
        [4]   // <fds
        [5].0   // DEFAULT
        [5].1   // NEW DEFAULT
        [6]   // ph vers venturi
        [9].1   // ack STOCK
        [20].0   // DEFAUT POSITION VANNE VENTURI
        [20].1   // defaut ultima pmp renvoi 1
        [20].2   // defaut ultima pmp renvoi 2
        [20].3   // présence pmp renvoi 1
        [20].4   // présence pmp renvoi 2
        [20].5   // ready drive pmp acide nautral
        [20].6   // ready drive pmp base neutral
        [20].7   // niveau bassin TOO HIGH
        [20].8   // ph vers venturi TOO HIGH
        [20].9   // ph vers venturi TOO LOW
        [20].10   // ph IN venturi TOO HIGH
        [20].11   // ph IN venturi TOO LOW
        [20].12   // FLOW VENTURI TOO HIGH
        [25].0   // DEFAUT POSITION VANNE VENTURI
        [25].1   // defaut ultima pmp renvoi 1
        [25].2   // defaut ultima pmp renvoi 2
        [25].3   // présence pmp renvoi 1
        [25].4   // présence pmp renvoi 2
        [25].5   // ready drive pmp acide nautral
        [25].6   // ready drive pmp base neutral
        [25].7   // niveau bassin TOO HIGH
        [25].8   // ph vers venturi TOO HIGH
        [25].9   // ph vers venturi TOO LOW
        [25].10   // ph IN venturi TOO HIGH
        [25].11   // ph IN venturi TOO LOW
        [25].12   // FLOW VENTURI TOO HIGH
        [30]   // NOMBRE DE DEFAUTS
        [31]   // MEMO NOMBRE DE DEFAUTS
   N7 : DINT[30] := ([3] := 49, [4] := 794, [6] := -79, [7] := -93, [8] := 151, [10] := 22575, [11] := 40, [20] := -75, [23] := 4);
        [3]   // aux. tot debit venturi
        [5]   // vitesse pmp Ph > 7
        [6]   // vitesse pmp Ph < 7
        [10]   // AUX. Consigne position vanne renvoi
        [20]   // dh-> ibt T°venturi
        [21]   // DEFAUT PRIORITE 1
        [22]   // DEFAUT PRIORITE 2
        [23]   // dh-> ibt
        [24]   // dh-> ibt
        [25]   // dh-> ibt
        [26]   // dh-> ibt
        [27]   // dh-> ibt
        [28]   // dh-> ibt
        [29]   // dh-> ibt
   N9 : DINT[50] := ([3] := 775, [4] := 600, [5] := 900, [6] := 580, [7] := 950, [8] := 790, [9] := 680, [10] := 605, [11] := 747, [12] := 41, [13] := 759, [14] := 30, [15] := 637, [16] := 12, [17] := -75, [18] := 70, [20] := 4103, [21] := 27, [22] := 10, [23] := 12, [24] := 137, [25] := 160, [28] := 5, [40] := 40);
        [3]   // ph vers venturi
        [4]   // histeresis low Ph venturi default venturi
        [5]   // histeresis high Ph venturi default venturi
        [6]   // Sp Ph venturi
        [10]   // position servo vanne renvoi
        [11]   // ph vers venturi
        [12]   // debit venturi
        [13]   // ph venturi
        [14]   // conduct venturi mS
        [15]   // ph neutral
        [16]   // niveau bassin
        [17]   // T°venturi
        [18]   // % ouverture vanne renvoi vers neutral
        [19]   // dsffds
        [20]   // msg vers ibt
   T4 : TIMER[25] := ([1].PRE := 10000, [1].ACC := 4850, [1].EN := 1, [1].TT := 1, [2].PRE := 10000, [2].ACC := 4850, [2].EN := 1, [2].TT := 1, [3].PRE := 60000, [3].ACC := 50650, [3].EN := 1, [3].TT := 1, [4].PRE := 60000, [4].ACC := 50650, [4].EN := 1, [4].TT := 1, [5].PRE := 180, [9].PRE := 180000, [9].ACC := 180000, [10].PRE := 300000, [11].PRE := 180000, [11].ACC := 180000, [19].PRE := 180000, [19].EN := 1, [19].DN := 1);
        [1]   // TEMPO 10 SEC
        [2]   // tempo envoi msg vers ibt
        [3]   // tempo 1 min
        [4]   // T 1 min
        [9]   // tempo off defaut PH vers venturi
        [10]   // tempo defaut PH vers venturi
        [11]   // tempo defaut ph venturi
        [19]   // DEFAUT POSITION VANNE VENTURI
END_VAR
